// TwinCAT 3 PLC project PLC1
// ProgramVersion: 3.1.4023.0
// libraries:
//   Tc2_EtherCAT, * (Beckhoff Automation GmbH)
//   Tc2_Standard, * (Beckhoff Automation GmbH)
//   Tc2_System, * (Beckhoff Automation GmbH)
//   Tc2_Utilities, * (Beckhoff Automation GmbH)
//   Tc3_Module, * (Beckhoff Automation GmbH)
// project tree:
//   DUTs/ DT_Incidence.TcDUT, DT_Incidences.TcDUT, DT_Incidence_Severity.TcDUT
//   GVLs/ OPC_UA.TcGVL
//   / PlcTask.TcTTO
//   POUs/ MAIN.TcPOU

CONFIGURATION PLC1
    RESOURCE PLC ON TwinCAT3
        TASK PlcTask(INTERVAL := T#10ms, PRIORITY := 20);
        PROGRAM MAIN WITH PlcTask : MAIN;
    END_RESOURCE
END_CONFIGURATION

// ---- DUTs/DT_Incidence.TcDUT
{attribute 'OPC.UA.DA' := '1'}
{attribute 'OPC.UA.DA.StructuredType' := '1'}
TYPE DT_Incidence :
	STRUCT
	//From Self Name
	WareHouse: STRING;
	Device: STRING;
	//Coded Value
	Id: STRING(10);
	//Exactly definition
	Description: STRING(255);
	Severity: DT_Incidence_Severity;
	//Cíclic Results
	State: BOOL;
	K: BOOL;
	END_STRUCT
END_TYPE

// ---- DUTs/DT_Incidences.TcDUT
{attribute 'qualified_only'}
TYPE DT_Incidences :
	{attribute 'OPC.UA.DA' := '1'}
	{attribute 'OPC.UA.DA.StructuredType' := '1'}
	STRUCT
			n: ARRAY[1..10] OF DT_Incidence; 
	END_STRUCT
END_TYPE

// ---- DUTs/DT_Incidence_Severity.TcDUT
{attribute 'qualified_only'}
{attribute 'strict'}
TYPE DT_Incidence_Severity :
(
	Unknown := 0,
	Warning	:= 1,
	Error	:= 2,
	Fatal	:= 3
);
END_TYPE

// ---- GVLs/OPC_UA.TcGVL
{attribute 'qualified_only'}
VAR_GLOBAL
	{attribute 'OPC.UA.DA' := '1'}
	{attribute 'OPC.UA.DA.StructuredType' := '1'}
	Alrm: DT_Incidences;

	
END_VAR

// ---- POUs/MAIN.TcPOU
PROGRAM MAIN

VAR
	bReconfig: BOOL := FALSE;
	bInit: BOOL := false;
END_VAR



A01_Init();

ACTION A01_Init:
IF NOT bInit OR bReconfig THEN 
	bReconfig:= FALSE;
			
	OPC_UA.Alrm.n[1].WareHouse:= '=MCP1';
	OPC_UA.Alrm.n[1].Device:= '-1Q1';
	OPC_UA.Alrm.n[1].Id:= '01920192';
	OPC_UA.Alrm.n[1].Description:= 'Main Switch';
	OPC_UA.Alrm.n[1].Severity:= DT_Incidence_Severity.Fatal;

	OPC_UA.Alrm.n[2].WareHouse:= '=MCP1';
	OPC_UA.Alrm.n[2].Device:= '-5F1';
	OPC_UA.Alrm.n[2].Id:= '02000200';
	OPC_UA.Alrm.n[2].Description:= 'Surge Arrester';
	OPC_UA.Alrm.n[2].Severity:= DT_Incidence_Severity.Error;

	OPC_UA.Alrm.n[3].WareHouse:= '=MCP1';
	OPC_UA.Alrm.n[3].Device:= '-9F1';
	OPC_UA.Alrm.n[3].Id:= '11001100';
	OPC_UA.Alrm.n[3].Description:= 'Circuit Breaker (AS-interface Power Supply 1)';
	OPC_UA.Alrm.n[3].Severity:= DT_Incidence_Severity.Fatal;
	
	OPC_UA.Alrm.n[4].WareHouse:= '=MCP1';
	OPC_UA.Alrm.n[4].Device:= '-9F2';
	OPC_UA.Alrm.n[4].Id:= '31003100';
	OPC_UA.Alrm.n[4].Description:= 'Photoeye Tripped';
	OPC_UA.Alrm.n[4].Severity:= DT_Incidence_Severity.Fatal;

	OPC_UA.Alrm.n[5].WareHouse:= '=MCP1';
	OPC_UA.Alrm.n[5].Device:= '-20F1';
	OPC_UA.Alrm.n[5].Id:= '42004200';
	OPC_UA.Alrm.n[5].Description:= 'Power Fuse (Power Distributor internal devices)';
	OPC_UA.Alrm.n[5].Severity:= DT_Incidence_Severity.Fatal;
	
	OPC_UA.Alrm.n[6].WareHouse:= '=MCP1';
	OPC_UA.Alrm.n[6].Device:= '-20F2';
	OPC_UA.Alrm.n[6].Id:= '02200220';
	OPC_UA.Alrm.n[6].Description:= 'Ethercat Bus Communication Lost';
	OPC_UA.Alrm.n[6].Severity:= DT_Incidence_Severity.Warning;

	OPC_UA.Alrm.n[7].WareHouse:= '=MCP1';
	OPC_UA.Alrm.n[7].Device:= '-21F1';
	OPC_UA.Alrm.n[7].Id:= '45674567';
	OPC_UA.Alrm.n[7].Description:= 'Power Fuse (Power Distributor external devices)';
	OPC_UA.Alrm.n[7].Severity:= DT_Incidence_Severity.Fatal;

	OPC_UA.Alrm.n[8].WareHouse:= '=MCP1';
	OPC_UA.Alrm.n[8].Device:= '-22F1';
	OPC_UA.Alrm.n[8].Id:= '32003200';
	OPC_UA.Alrm.n[8].Description:= 'Photoeye Trigger';
	OPC_UA.Alrm.n[8].Severity:= DT_Incidence_Severity.Error;

	OPC_UA.Alrm.n[9].WareHouse:= '=MCP1';
	OPC_UA.Alrm.n[9].Device:= '-26K1';
	OPC_UA.Alrm.n[9].Id:= '74837483';
	OPC_UA.Alrm.n[9].Description:= 'FeedBack System (Area =CA1 & =CA2)';
	OPC_UA.Alrm.n[9].Severity:= DT_Incidence_Severity.Fatal;

	OPC_UA.Alrm.n[10].WareHouse:= '=MCP1';
	OPC_UA.Alrm.n[10].Device:= '-24K1';
	OPC_UA.Alrm.n[10].Id:= '38333833';
	OPC_UA.Alrm.n[10].Description:= 'FeedBack System Delayed (Area =CA1 & =CA2)';
	OPC_UA.Alrm.n[10].Severity:= DT_Incidence_Severity.Fatal;
END_IF
END_ACTION

END_PROGRAM
